// TIA Portal project "Proyecto_Final" (V18)

(* hardware
DEVICE "S7-1500/ET200MP station_1"  S7-1500 station
   slot 0: "Rail_0"  Rack  6ES7 590-1***0-0AA0
   slot 1: "PLC_1"  CPU 1511-1 PN  6ES7 511-1AK00-0AB0  V1.0
      slot 3: "CPU display_1"  6ES7591-1XA00-0AA0
      slot 32768: "PROFINET interface_1"  X1
   slot 2: "CM 1542-5_1"  CM 1542-5  6GK7 542-5DX00-0XE0  V1.0
   slot 3: "DI 16x24VDC HF_1"  DI 16x24VDC HF  6ES7 521-1BH00-0AB0  V1.0
   slot 4: "DQ 16x24VDC/0.5A ST_1"  DQ 16x24VDC/0.5A ST  6ES7 522-1BH00-0AB0  V2.0
   slot 5: "AI 8xU/I/RTD/TC ST_1"  AI 8xU/I/RTD/TC ST  6ES7 531-7KF00-0AB0  V1.0
   slot 6: "AQ 4xU/I ST_1"  AQ 4xU/I ST  6ES7 532-5HD00-0AB0  V1.0
DEVICE "HMI_1"  KTP600 Basic color PN
   slot 0: "HMI_1"  KTP600 Basic color PN  6AV6 647-0AD11-3AX0  12.0.0.0
   slot 1: "HMI_RT_1"  KTP600 Basic color PN  6AV6 647-0AD11-3AX0  12.0.0.0
   slot 5: "HMI_1.IE_CP_1"  PROFINET Interface  12.0.0.0
      slot 1: "PROFINET Interface_1"  PROFINET Interface
         slot 1: "Port_1"  Port
DEVICE "PC-System_1"  SIMATIC PC station
   slot 0: "SIMATIC PC station"  Rail  SIMATIC PC-Station  V1.0
      slot 125: "Stationmanager"  Station_Manager  V6.0.4
   slot 1: "HMI_RT_2"  WinCC RT Advanced  6AV2 104-0xxxx-xxxx  17.0.0.0
      slot 33792: "Computer interface"  Host interface
   slot 2: "IE general_1"  IE General  IE_CP  V8.2.0
      slot 1: "PROFINET interface"  IEGeneral.Interface.8.2.0
*)

// ===== PLC "PLC_1"  CPU 1511-1 PN =====

VAR_GLOBAL   // PLC tag table "Default tag table"
   "Start" AT %M3.4 : Bool;
   "Stop" AT %M3.5 : Bool;
   "PE" AT %M3.6 : Bool;
   "Motor_Banda" AT %Q0.0 : Bool;
   "Variador_Metal" AT %Q0.1 : Bool;
   "V_Presencia" AT %I0.3 : Bool;
   "Reset" AT %M0.0 : Bool;
   "V_Sensor_Metal" AT %I0.4 : Bool;
   "V_Sensor_Vidrio" AT %I0.6 : Bool;
   "V_Galga" AT %IW2 : Int;
   "Medir" AT %M0.1 : Bool;
   "Metal" AT %M0.2 : Bool;
   "Vidrio" AT %M0.3 : Bool;
   "Plastico" AT %M0.4 : Bool;
   "Temp_1s" AT %M0.5 : Bool;
   "T1s_OK" AT %M0.6 : Bool;
   "CTU_Metal" AT %M0.7 : Bool;
   "Metal_OK" AT %M1.0 : Bool;
   "CTU_Vidrio" AT %M1.1 : Bool;
   "Vidrio_OK" AT %M1.2 : Bool;
   "CTU_Plastico" AT %M1.3 : Bool;
   "Plastico_OK" AT %M1.4 : Bool;
   "Temp_Peso" AT %M1.5 : Bool;
   "Temp_Peso_OK" AT %M1.6 : Bool;
   "PID_Pesaje" AT %M1.7 : Bool;
   "Temp_3s" AT %M2.0 : Bool;
   "T3s_OK" AT %M2.1 : Bool;
   "Peso" AT %M2.2 : Bool;
   "Temp_7s" AT %M2.3 : Bool;
   "T7s_OK" AT %M2.4 : Bool;
   "Temp_5s" AT %M2.5 : Bool;
   "T5s_OK" AT %M2.6 : Bool;
   "Temp_Variador" AT %M2.7 : Bool;
   "Temp_Vari_OK" AT %M3.0 : Bool;
   "R_Metal" AT %M3.1 : Bool;
   "R_Vidrio" AT %M3.2 : Bool;
   "R_Plastico" AT %M3.3 : Bool;
   "Piston_Plastico" AT %Q0.2 : Bool;
   "Start_Fisico" AT %I0.0 : Bool;
   "Stop_Fisico" AT %I0.1 : Bool;
   "PE_Fisico" AT %I0.2 : Bool;
   "Start_Pulse" AT %Q0.3 : Bool;
   "En_Pulse" AT %M4.0 : Bool;
   "Low_Pulse_Active" AT %M4.1 : Bool;
   "High_Pulse_Enable" AT %M4.2 : Bool;
   "High_Pulse_Active" AT %M4.3 : Bool;
   "Low_Pulse_Enable" AT %M4.4 : Bool;
   "Count_Metal" AT %QD100 : Real;
   "Count_Vidrio" AT %QD108 : Real;
   "Count_Plastico" AT %QD104 : Real;
   "Alarma_StartNoPresence" AT %Q1.1 : Bool;
   "Alarma_Inicio" AT %Q1.2 : Bool;
   "Alarma_Final" AT %Q1.3 : Bool;
   "Alarma_PE" AT %Q1.0 : Bool;
   "aux" AT %M20.0 : Bool;
   "Start_Fisico_old" AT %M10.4 : Bool;
   "Material_Detectado" AT %Q1.4 : Bool;
   "STP_FIO" AT %I20.1 : Bool;
   "PE_FIO" AT %I20.2 : Bool;
   "START_FIO" AT %I20.0 : Bool;
   "Stop_HMI" AT %M30.1 : Bool;
   "PE_HMI" AT %M30.2 : Bool;
   "START_HMI" AT %M30.3 : Bool;
   "Receta_1" AT %M30.4 : Bool;
   "R1" AT %M30.5 : Bool;
   "R2" AT %M30.6 : Bool;
   "Receta_2" AT %M30.7 : Bool;
END_VAR

DATA_BLOCK "Block_2_DB"   // DB10
{ S7_Optimized_Access := 'TRUE' }
VERSION : 0.1
// stored: InstanceOfName Block_2
"Block_2"
BEGIN
END_DATA_BLOCK

DATA_BLOCK "Block_1_DB"   // DB11
{ S7_Optimized_Access := 'TRUE' }
VERSION : 0.1
// stored: InstanceOfName Grafcet
"Grafcet"
BEGIN
END_DATA_BLOCK

// folder: System blocks/Program resources

DATA_BLOCK "IEC_Timer_0_DB"   // DB1
{ S7_Optimized_Access := 'TRUE' }
AUTHOR : Simatic
FAMILY : IEC
NAME : IEC_TMR
VERSION : 1.0
// stored: InstanceOfName IEC_TIMER
"IEC_TIMER"
BEGIN
END_DATA_BLOCK

DATA_BLOCK "IEC_Counter_0_DB"   // DB2
{ S7_Optimized_Access := 'TRUE' }
AUTHOR : Simatic
FAMILY : IEC
NAME : CNTR
VERSION : 1.0
// stored: InstanceOfName IEC_COUNTER
"IEC_COUNTER"
BEGIN
END_DATA_BLOCK

DATA_BLOCK "IEC_Counter_0_DB_1"   // DB3
{ S7_Optimized_Access := 'TRUE' }
AUTHOR : Simatic
FAMILY : IEC
NAME : CNTR
VERSION : 1.0
// stored: InstanceOfName IEC_COUNTER
"IEC_COUNTER"
BEGIN
END_DATA_BLOCK

DATA_BLOCK "IEC_Counter_0_DB_2"   // DB4
{ S7_Optimized_Access := 'TRUE' }
AUTHOR : Simatic
FAMILY : IEC
NAME : CNTR
VERSION : 1.0
// stored: InstanceOfName IEC_COUNTER
"IEC_COUNTER"
BEGIN
END_DATA_BLOCK

DATA_BLOCK "IEC_Timer_0_DB_1"   // DB5
{ S7_Optimized_Access := 'TRUE' }
AUTHOR : Simatic
FAMILY : IEC
NAME : IEC_TMR
VERSION : 1.0
// stored: InstanceOfName IEC_TIMER
"IEC_TIMER"
BEGIN
END_DATA_BLOCK

DATA_BLOCK "IEC_Timer_0_DB_2"   // DB6
{ S7_Optimized_Access := 'TRUE' }
AUTHOR : Simatic
FAMILY : IEC
NAME : IEC_TMR
VERSION : 1.0
// stored: InstanceOfName IEC_TIMER
"IEC_TIMER"
BEGIN
END_DATA_BLOCK

DATA_BLOCK "IEC_Timer_0_DB_3"   // DB7
{ S7_Optimized_Access := 'TRUE' }
AUTHOR : Simatic
FAMILY : IEC
NAME : IEC_TMR
VERSION : 1.0
// stored: InstanceOfName IEC_TIMER
"IEC_TIMER"
BEGIN
END_DATA_BLOCK

DATA_BLOCK "IEC_Timer_0_DB_4"   // DB8
{ S7_Optimized_Access := 'TRUE' }
AUTHOR : Simatic
FAMILY : IEC
NAME : IEC_TMR
VERSION : 1.0
// stored: InstanceOfName IEC_TIMER
"IEC_TIMER"
BEGIN
END_DATA_BLOCK

DATA_BLOCK "IEC_Timer_0_DB_5"   // DB9
{ S7_Optimized_Access := 'TRUE' }
AUTHOR : Simatic
FAMILY : IEC
NAME : IEC_TMR
VERSION : 1.0
// stored: InstanceOfName IEC_TIMER
"IEC_TIMER"
BEGIN
END_DATA_BLOCK

// folder: (top level)

FUNCTION_BLOCK "Grafcet"   // FB1, GRAPH_PLUS
{ S7_Optimized_Access := 'TRUE' }
VERSION : 0.1
   VAR_INPUT
      OFF_SQ : Bool := false;   // Turn sequence off
      INIT_SQ : Bool := false;   // Set sequence to initial state
      ACK_EF : Bool := false;   // Acknowledge all errors and faults
      S_PREV : Bool := false;   // Output previous step in parameter S_NO
      S_NEXT : Bool := false;   // Indicate next step in parameter S_NO
      SW_AUTO : Bool := false;   // Automatic mode
      SW_TAP : Bool := false;   // Semiautomatic/switch with transition
      SW_TOP : Bool := false;   // Semiautomatic/ignore transition
      SW_MAN : Bool := false;   // Manual mode
      S_SEL : Int := 0;   // Select step to be output to S_NO
      S_ON : Bool := false;   // Activate step indicated in S_NO
      S_OFF : Bool := false;   // Disable step indicated in S_NO
      T_PUSH : Bool := false;   // Enable transition to switch in semi automatic mode
   END_VAR
   VAR_OUTPUT
      S_NO : Int := 0;   // Step number
      S_MORE : Bool := false;   // More steps are available and can be shown in S_NO
      S_ACTIVE : Bool := false;   // Step indicated in S_NO is active
      ERR_FLT : Bool := false;   // Interlock or supervision group error
      AUTO_ON : Bool := false;   // Automatic mode is active
      TAP_ON : Bool := false;   // Semiautomatic mode/step with transition enabled
      TOP_ON : Bool := false;   // Semiautomatic mode/ignore transition enabled
      MAN_ON : Bool := false;   // Manual mode is active
   END_VAR
   VAR
      HMI_INFO : Array[0..8] of UInt;
      IF_PAR : G7_IfParPlus_V2;
      RT_DATA : G7_RTDataPlus_V2;   // Internal data area
      Trans1 : G7_TransitionPlus_V2;   // Transition structure
      Trans5 : G7_TransitionPlus_V2;   // Transition structure
      Trans7 : G7_TransitionPlus_V2;   // Transition structure
      Trans8 : G7_TransitionPlus_V2;   // Transition structure
      Trans9 : G7_TransitionPlus_V2;   // Transition structure
      Trans10 : G7_TransitionPlus_V2;   // Transition structure
      Trans11 : G7_TransitionPlus_V2;   // Transition structure
      Trans12 : G7_TransitionPlus_V2;   // Transition structure
      Trans13 : G7_TransitionPlus_V2;   // Transition structure
      Trans14 : G7_TransitionPlus_V2;   // Transition structure
      Trans15 : G7_TransitionPlus_V2;   // Transition structure
      Trans16 : G7_TransitionPlus_V2;   // Transition structure
      Trans17 : G7_TransitionPlus_V2;   // Transition structure
      Trans18 : G7_TransitionPlus_V2;   // Transition structure
      Trans19 : G7_TransitionPlus_V2;   // Transition structure
      Trans20 : G7_TransitionPlus_V2;   // Transition structure
      Trans21 : G7_TransitionPlus_V2;   // Transition structure
      Trans22 : G7_TransitionPlus_V2;   // Transition structure
      Trans23 : G7_TransitionPlus_V2;   // Transition structure
      Trans24 : G7_TransitionPlus_V2;   // Transition structure
      Trans26 : G7_TransitionPlus_V2;   // Transition structure
      Trans27 : G7_TransitionPlus_V2;   // Transition structure
      Trans28 : G7_TransitionPlus_V2;   // Transition structure
      Trans29 : G7_TransitionPlus_V2;   // Transition structure
      Trans30 : G7_TransitionPlus_V2;   // Transition structure
      Trans31 : G7_TransitionPlus_V2;   // Transition structure
      Reset : G7_StepPlus_V2;   // Step structure
      "Ingreso Botella" : G7_StepPlus_V2;   // Step structure
      Avance_Banda : G7_StepPlus_V2;   // Step structure
      Pesaje : G7_StepPlus_V2;   // Step structure
      Pos_Metal : G7_StepPlus_V2;   // Step structure
      Contenedor_Metal : G7_StepPlus_V2;   // Step structure
      Fin_Ciclo_Metal : G7_StepPlus_V2;   // Step structure
      Pos_Vidrio : G7_StepPlus_V2;   // Step structure
      Contenedor_Vidrio : G7_StepPlus_V2;   // Step structure
      Fin_Ciclo_Vidrio : G7_StepPlus_V2;   // Step structure
      Pos_Plastico : G7_StepPlus_V2;   // Step structure
      Contenedor_Plastico : G7_StepPlus_V2;   // Step structure
      Fin_Ciclo_Plastico : G7_StepPlus_V2;   // Step structure
      Alarmas : G7_StepPlus_V2;   // Step structure
      Step16 : G7_StepPlus_V2;   // Step structure
      Contenedor_Vidrio_1 : G7_StepPlus_V2;   // Step structure
      Alarmas1 : G7_StepPlus_V2;   // Step structure
      Alarmas3 : G7_StepPlus_V2;   // Step structure
      Step20 : G7_StepPlus_V2;   // Step structure
      SINI : Array[0..1] of USInt;
      LSTT : Array[0..25] of USInt;
      ATAJ : Array[0..25] of USInt;
      ATAB : Array[0..25] of USInt;
      PSTT : Array[0..25] of USInt;
      NSTT : Array[0..25] of USInt;
      ASSJ : Array[0..18] of USInt;
      ASSB : Array[0..18] of USInt;
      PTTS : Array[0..18] of USInt;
      NTTS : Array[0..18] of USInt;
      SW_SQTS : Array[0..18] of USInt;
      SWITCH : Array[0..15] of USInt;
      TVX : Array[0..14] of USInt;
      TTX : Array[0..14] of USInt;
      TSX : Array[0..1] of USInt;
      S00X : Array[0..1] of USInt;
      SOFFX : Array[0..1] of USInt;
      SONX : Array[0..1] of USInt;
      SAX : Array[0..1] of USInt;
      SERRX : Array[0..19] of USInt;
      SMX : Array[0..19] of USInt;
      S0X : Array[0..19] of USInt;
      S1X : Array[0..19] of USInt;
      IL_ALARM_INST : Program_Alarm;
      SUP_ALARM_INST : Program_Alarm;
      STEP_TIME_ALARM_INST : Program_Alarm;
      IEC_TIMER_INST : IEC_TIMER;
      TRANSACTION_FLAG : Bool := false;
   END_VAR
   // SINI[0] := 2;
   // LSTT[0] := 255;
   // LSTT[1] := 255;
   // LSTT[2] := 255;
   // LSTT[3] := 255;
   // LSTT[4] := 255;
   // LSTT[5] := 255;
   // LSTT[6] := 255;
   // LSTT[7] := 255;
   // LSTT[8] := 255;
   // LSTT[9] := 1;
   // LSTT[10] := 255;
   // LSTT[11] := 255;
   // LSTT[12] := 1;
   // LSTT[13] := 255;
   // LSTT[14] := 255;
   // LSTT[15] := 255;
   // LSTT[16] := 1;
   // LSTT[17] := 255;
   // LSTT[19] := 255;
   // ATAJ[1] := 1;
   // ATAJ[2] := 2;
   // ATAJ[3] := 3;
   // ATAJ[4] := 4;
   // ATAJ[5] := 5;
   // ATAJ[6] := 6;
   // ATAJ[7] := 7;
   // ATAJ[8] := 8;
   // ATAJ[9] := 9;
   // ATAJ[10] := 10;
   // ATAJ[11] := 11;
   // ATAJ[12] := 12;
   // ATAJ[13] := 13;
   // ATAJ[14] := 14;
   // ATAJ[15] := 15;
   // ATAJ[16] := 16;
   // ATAJ[17] := 17;
   // ATAJ[18] := 18;
   // ATAJ[19] := 19;
   // ATAJ[20] := 20;
   // ATAJ[21] := 21;
   // ATAB[1] := 1;
   // ATAB[2] := 2;
   // ATAB[3] := 4;
   // ATAB[4] := 5;
   // ATAB[5] := 3;
   // ATAB[6] := 22;
   // ATAB[7] := 7;
   // ATAB[8] := 9;
   // ATAB[9] := 8;
   // ATAB[10] := 24;
   // ATAB[11] := 11;
   // ATAB[12] := 13;
   // ATAB[13] := 12;
   // ATAB[14] := 14;
   // ATAB[15] := 15;
   // ATAB[16] := 17;
   // ATAB[17] := 16;
   // ATAB[18] := 18;
   // ATAB[19] := 19;
   // ATAB[20] := 20;
   // ATAB[21] := 21;
   // PSTT[1] := 1;
   // PSTT[2] := 2;
   // PSTT[3] := 3;
   // PSTT[4] := 3;
   // PSTT[5] := 3;
   // PSTT[6] := 4;
   // PSTT[7] := 5;
   // PSTT[8] := 6;
   // PSTT[9] := 6;
   // PSTT[10] := 7;
   // PSTT[11] := 8;
   // PSTT[12] := 9;
   // PSTT[13] := 9;
   // PSTT[14] := 10;
   // PSTT[15] := 11;
   // PSTT[16] := 12;
   // PSTT[17] := 12;
   // PSTT[18] := 13;
   // PSTT[19] := 14;
   // PSTT[20] := 16;
   // PSTT[21] := 17;
   // NSTT[0] := 1;
   // NSTT[1] := 2;
   // NSTT[2] := 3;
   // NSTT[3] := 4;
   // NSTT[4] := 7;
   // NSTT[5] := 10;
   // NSTT[6] := 5;
   // NSTT[7] := 6;
   // NSTT[8] := 13;
   // NSTT[9] := 1;
   // NSTT[10] := 8;
   // NSTT[11] := 9;
   // NSTT[12] := 1;
   // NSTT[13] := 14;
   // NSTT[14] := 11;
   // NSTT[15] := 12;
   // NSTT[16] := 1;
   // NSTT[17] := 17;
   // NSTT[19] := 16;
   // ASSJ[1] := 1;
   // ASSJ[2] := 2;
   // ASSJ[3] := 3;
   // ASSJ[4] := 4;
   // ASSJ[5] := 5;
   // ASSJ[6] := 6;
   // ASSJ[7] := 7;
   // ASSJ[8] := 8;
   // ASSJ[9] := 9;
   // ASSJ[10] := 10;
   // ASSJ[11] := 11;
   // ASSJ[12] := 12;
   // ASSJ[13] := 13;
   // ASSJ[14] := 14;
   // ASSJ[15] := 15;
   // ASSJ[16] := 16;
   // ASSB[1] := 1;
   // ASSB[2] := 2;
   // ASSB[3] := 3;
   // ASSB[4] := 4;
   // ASSB[5] := 5;
   // ASSB[6] := 6;
   // ASSB[7] := 7;
   // ASSB[8] := 8;
   // ASSB[9] := 9;
   // ASSB[10] := 10;
   // ASSB[11] := 11;
   // ASSB[12] := 12;
   // ASSB[13] := 13;
   // ASSB[14] := 14;
   // ASSB[15] := 15;
   // ASSB[16] := 16;
   // PTTS[0] := 255;
   // PTTS[2] := 1;
   // PTTS[3] := 2;
   // PTTS[4] := 3;
   // PTTS[5] := 6;
   // PTTS[6] := 7;
   // PTTS[7] := 4;
   // PTTS[8] := 10;
   // PTTS[9] := 11;
   // PTTS[10] := 5;
   // PTTS[11] := 14;
   // PTTS[12] := 15;
   // PTTS[13] := 8;
   // PTTS[14] := 13;
   // PTTS[15] := 24;
   // PTTS[16] := 19;
   // NTTS[1] := 1;
   // NTTS[2] := 2;
   // NTTS[3] := 3;
   // NTTS[4] := 6;
   // NTTS[5] := 7;
   // NTTS[6] := 9;
   // NTTS[7] := 10;
   // NTTS[8] := 11;
   // NTTS[9] := 12;
   // NTTS[10] := 14;
   // NTTS[11] := 15;
   // NTTS[12] := 16;
   // NTTS[13] := 18;
   // NTTS[14] := 19;
   // NTTS[15] := 25;
   // NTTS[16] := 20;
   // SW_SQTS[4] := 1;
   // SW_SQTS[5] := 2;
   // SW_SQTS[6] := 2;
   // SW_SQTS[7] := 3;
   // SW_SQTS[8] := 4;
   // SW_SQTS[9] := 4;
   // SW_SQTS[10] := 5;
   // SW_SQTS[11] := 5;
   // SW_SQTS[12] := 5;
   // SW_SQTS[13] := 6;
   // SW_SQTS[14] := 7;
   // SW_SQTS[15] := 8;
   // SW_SQTS[16] := 7;
   // TVX[0] := 16#1;
   // TTX[0] := 16#1;
   // TSX[0] := 16#1;
   // S00X[0] := 16#1;
   // SOFFX[0] := 16#1;
   // SONX[0] := 16#1;
   // SAX[0] := 16#1;
   // SERRX[0] := 16#1;
   // SMX[0] := 16#1;
   // S0X[0] := 16#1;
   // S1X[0] := 16#1;
   // LSTT[22] := 255;
   // LSTT[23] := 6;
   // LSTT[24] := 255;
   // LSTT[25] := 9;
   // ATAJ[22] := 22;
   // ATAJ[23] := 23;
   // ATAJ[24] := 24;
   // ATAJ[25] := 25;
   // ATAB[22] := 6;
   // ATAB[23] := 23;
   // ATAB[24] := 10;
   // ATAB[25] := 25;
   // PSTT[22] := 4;
   // PSTT[23] := 18;
   // PSTT[24] := 7;
   // PSTT[25] := 15;
   // NSTT[22] := 18;
   // NSTT[23] := 6;
   // NSTT[24] := 15;
   // NSTT[25] := 9;
   // ASSJ[17] := 17;
   // ASSJ[18] := 18;
   // ASSB[17] := 17;
   // ASSB[18] := 18;
   // PTTS[17] := 17;
   // PTTS[18] := 22;
   // NTTS[17] := 21;
   // NTTS[18] := 23;
   // SW_SQTS[17] := 9;
   // SW_SQTS[18] := 10;
BEGIN
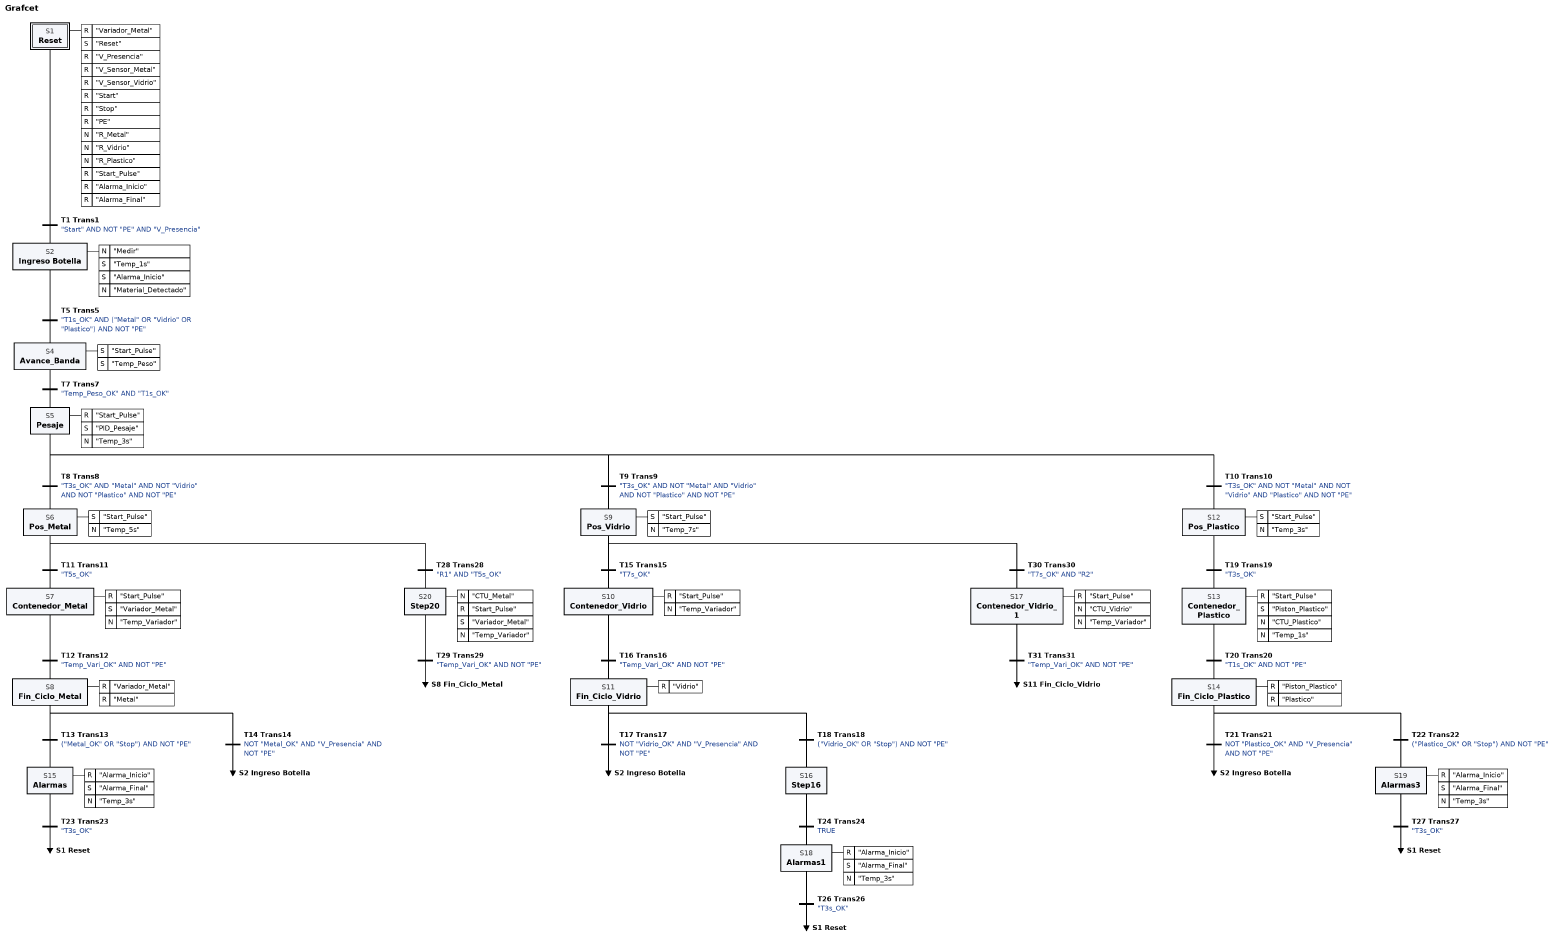
   // sequencer 1
   INITIAL_STEP Reset:   // S1, max time T#10S, warning time T#7S
              R    "Variador_Metal"
              S    "Reset"
              R    "V_Presencia"
              R    "V_Sensor_Metal"
              R    "V_Sensor_Vidrio"
              R    "Start"
              R    "Stop"
              R    "PE"
              N    "R_Metal"
              N    "R_Vidrio"
              N    "R_Plastico"
              R    "Start_Pulse"
              R    "Alarma_Inicio"
              R    "Alarma_Final"
              R    "Receta_1"
              R    "Receta_2"
              R    "R1"
              R    "R2"
   END_STEP
   TRANSITION Trans1 FROM Reset TO "Ingreso Botella"   // T1
      := "Start" AND NOT "PE" AND "V_Presencia";
   END_TRANSITION
   STEP "Ingreso Botella":   // S2, max time T#10S, warning time T#7S
              N    "Medir"
              S    "Temp_1s"
              S    "Alarma_Inicio"
              N    "Material_Detectado"
   END_STEP
   TRANSITION Trans5 FROM "Ingreso Botella" TO Avance_Banda   // T5
      := "T1s_OK" AND ("Metal" OR "Vidrio" OR "Plastico") AND NOT "PE";
   END_TRANSITION
   STEP Avance_Banda:   // S4, max time T#10S, warning time T#7S
              S    "Start_Pulse"
              S    "Temp_Peso"
   END_STEP
   TRANSITION Trans7 FROM Avance_Banda TO Pesaje   // T7
      := "Temp_Peso_OK" AND "T1s_OK";
   END_TRANSITION
   STEP Pesaje:   // S5, max time T#10S, warning time T#7S
              R    "Start_Pulse"
              S    "PID_Pesaje"
              N    "Temp_3s"
   END_STEP
   TRANSITION Trans8 FROM Pesaje TO Pos_Metal   // T8
      := "T3s_OK" AND "Metal" AND NOT "Vidrio" AND NOT "Plastico" AND NOT "PE";
   END_TRANSITION
   TRANSITION Trans9 FROM Pesaje TO Pos_Vidrio   // T9
      := "T3s_OK" AND NOT "Metal" AND "Vidrio" AND NOT "Plastico" AND NOT "PE";
   END_TRANSITION
   TRANSITION Trans10 FROM Pesaje TO Pos_Plastico   // T10
      := "T3s_OK" AND NOT "Metal" AND NOT "Vidrio" AND "Plastico" AND NOT "PE";
   END_TRANSITION
   STEP Pos_Metal:   // S6, max time T#10S, warning time T#7S
              S    "Start_Pulse"
              N    "Temp_5s"
   END_STEP
   TRANSITION Trans11 FROM Pos_Metal TO Contenedor_Metal   // T11
      := "T5s_OK";
   END_TRANSITION
   TRANSITION Trans28 FROM Pos_Metal TO Step20   // T28
      := "R1" AND "T5s_OK";
   END_TRANSITION
   STEP Contenedor_Metal:   // S7, max time T#10S, warning time T#7S
              R    "Start_Pulse"
              S    "Variador_Metal"
              N    "Temp_Variador"
   END_STEP
   TRANSITION Trans12 FROM Contenedor_Metal TO Fin_Ciclo_Metal   // T12
      := "Temp_Vari_OK" AND NOT "PE";
   END_TRANSITION
   STEP Fin_Ciclo_Metal:   // S8, max time T#10S, warning time T#7S
              R    "Variador_Metal"
              R    "Metal"
   END_STEP
   TRANSITION Trans13 FROM Fin_Ciclo_Metal TO Alarmas   // T13
      := ("Metal_OK" OR "Stop") AND NOT "PE";
   END_TRANSITION
   TRANSITION Trans14 FROM Fin_Ciclo_Metal TO "Ingreso Botella"   // T14, jump
      := NOT "Metal_OK" AND "V_Presencia" AND NOT "PE";
   END_TRANSITION
   STEP Pos_Vidrio:   // S9, max time T#10S, warning time T#7S
              S    "Start_Pulse"
              N    "Temp_7s"
   END_STEP
   TRANSITION Trans15 FROM Pos_Vidrio TO Contenedor_Vidrio   // T15
      := "T7s_OK";
   END_TRANSITION
   TRANSITION Trans30 FROM Pos_Vidrio TO Contenedor_Vidrio_1   // T30
      := "T7s_OK" AND "R2";
   END_TRANSITION
   STEP Contenedor_Vidrio:   // S10, max time T#10S, warning time T#7S
              R    "Start_Pulse"
              N    "Temp_Variador"
   END_STEP
   TRANSITION Trans16 FROM Contenedor_Vidrio TO Fin_Ciclo_Vidrio   // T16
      := "Temp_Vari_OK" AND NOT "PE";
   END_TRANSITION
   STEP Fin_Ciclo_Vidrio:   // S11, max time T#10S, warning time T#7S
              R    "Vidrio"
   END_STEP
   TRANSITION Trans17 FROM Fin_Ciclo_Vidrio TO "Ingreso Botella"   // T17, jump
      := NOT "Vidrio_OK" AND "V_Presencia" AND NOT "PE";
   END_TRANSITION
   TRANSITION Trans18 FROM Fin_Ciclo_Vidrio TO Step16   // T18
      := ("Vidrio_OK" OR "Stop") AND NOT "PE";
   END_TRANSITION
   STEP Pos_Plastico:   // S12, max time T#10S, warning time T#7S
              S    "Start_Pulse"
              N    "Temp_3s"
   END_STEP
   TRANSITION Trans19 FROM Pos_Plastico TO Contenedor_Plastico   // T19
      := "T3s_OK";
   END_TRANSITION
   STEP Contenedor_Plastico:   // S13, max time T#10S, warning time T#7S
              R    "Start_Pulse"
              S    "Piston_Plastico"
              N    "CTU_Plastico"
              N    "Temp_1s"
   END_STEP
   TRANSITION Trans20 FROM Contenedor_Plastico TO Fin_Ciclo_Plastico   // T20
      := "T1s_OK" AND NOT "PE";
   END_TRANSITION
   STEP Fin_Ciclo_Plastico:   // S14, max time T#10S, warning time T#7S
              R    "Piston_Plastico"
              R    "Plastico"
   END_STEP
   TRANSITION Trans21 FROM Fin_Ciclo_Plastico TO "Ingreso Botella"   // T21, jump
      := NOT "Plastico_OK" AND "V_Presencia" AND NOT "PE";
   END_TRANSITION
   TRANSITION Trans22 FROM Fin_Ciclo_Plastico TO Alarmas3   // T22
      := ("Plastico_OK" OR "Stop") AND NOT "PE";
   END_TRANSITION
   STEP Alarmas:   // S15, max time T#10S, warning time T#7S
              R    "Alarma_Inicio"
              S    "Alarma_Final"
              N    "Temp_3s"
   END_STEP
   TRANSITION Trans23 FROM Alarmas TO Reset   // T23, jump
      := "T3s_OK";
   END_TRANSITION
   STEP Step16:   // S16, max time T#10S, warning time T#7S
   END_STEP
   TRANSITION Trans24 FROM Step16 TO Alarmas1   // T24
      := TRUE;
   END_TRANSITION
   STEP Alarmas1:   // S18, max time T#10S, warning time T#7S
              R    "Alarma_Inicio"
              S    "Alarma_Final"
              N    "Temp_3s"
   END_STEP
   TRANSITION Trans26 FROM Alarmas1 TO Reset   // T26, jump
      := "T3s_OK";
   END_TRANSITION
   STEP Alarmas3:   // S19, max time T#10S, warning time T#7S
              R    "Alarma_Inicio"
              S    "Alarma_Final"
              N    "Temp_3s"
   END_STEP
   TRANSITION Trans27 FROM Alarmas3 TO Reset   // T27, jump
      := "T3s_OK";
   END_TRANSITION
   STEP Step20:   // S20, max time T#10S, warning time T#7S
              N    "CTU_Metal"
              R    "Start_Pulse"
              S    "Variador_Metal"
              N    "Temp_Variador"
   END_STEP
   TRANSITION Trans29 FROM Step20 TO Fin_Ciclo_Metal   // T29, jump
      := "Temp_Vari_OK" AND NOT "PE";
   END_TRANSITION
   STEP Contenedor_Vidrio_1:   // S17, max time T#10S, warning time T#7S
              R    "Start_Pulse"
              N    "CTU_Vidrio"
              N    "Temp_Variador"
   END_STEP
   TRANSITION Trans31 FROM Contenedor_Vidrio_1 TO Fin_Ciclo_Vidrio   // T31, jump
      := "Temp_Vari_OK" AND NOT "PE";
   END_TRANSITION
END_FUNCTION_BLOCK

FUNCTION_BLOCK "Block_2"   // FB2, STL
{ S7_Optimized_Access := 'TRUE' }
VERSION : 0.1
   VAR
      IEC_Timer_0_Instance : TON_LTIME;
      DB1 : TON_LTIME;
   END_VAR
BEGIN

REGION Network 1
   // Habilitación
         A     "Start_Pulse";
         =     "En_Pulse";

   // Enable T1
         A     "En_Pulse";
         AN    "Low_Pulse_Active";
         =     "High_Pulse_Enable";

         CALL  #DB1
         ( IN := "High_Pulse_Enable",
           PT := LT#25000ns,
           Q  := "High_Pulse_Active",
           ET :=
         );


   // Enable T2
         A     "En_Pulse";
         A     "High_Pulse_Active";
         =     "Low_Pulse_Enable";

         CALL  #IEC_Timer_0_Instance
         ( IN := "Low_Pulse_Enable",
           PT := LT#25000ns,
           Q  := "Low_Pulse_Active",
           ET :=
         );

   // Salida
         A     "High_Pulse_Active";
         =     "Motor_Banda";
END_REGION
END_FUNCTION_BLOCK

ORGANIZATION_BLOCK "Main"   // OB1, LAD, ProgramCycle
TITLE = "Main Program Sweep (Cycle)"
{ S7_Optimized_Access := 'TRUE' }
VERSION : 0.1
   VAR_INPUT
      Initial_Call : Bool;   // Initial call of this OB
      Remanence : Bool;   // =True, if remanent data are available
   END_VAR
BEGIN

REGION Network 1
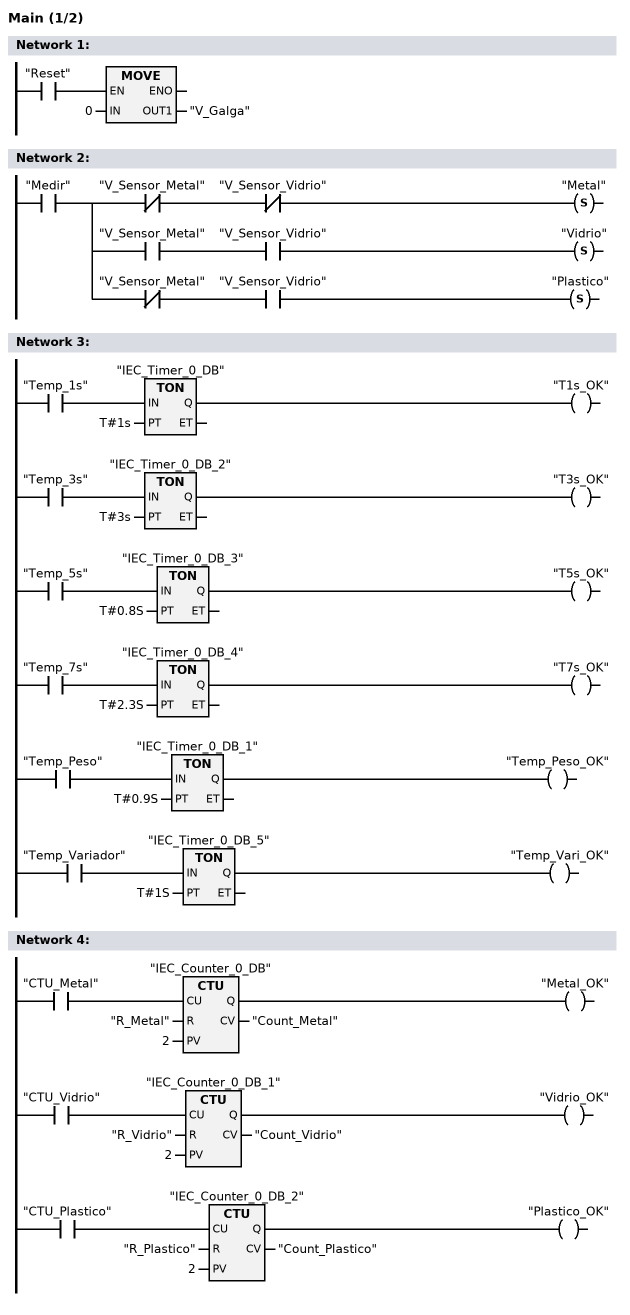
   RUNG wire#powerrail
      Contact( "Reset" )
      Move(in := 0, out1 => "V_Galga")
   END_RUNG
   // the same network as SCL:
   IF "Reset" THEN "V_Galga" := 0; END_IF;
END_REGION

REGION Network 2
   RUNG wire#powerrail
      Contact( "Medir" )
      wire#w1
      I_Contact( "V_Sensor_Metal" )
      I_Contact( "V_Sensor_Vidrio" )
      S_Coil( "Metal" )
   END_RUNG
   RUNG wire#w1
      Contact( "V_Sensor_Metal" )
      Contact( "V_Sensor_Vidrio" )
      S_Coil( "Vidrio" )
   END_RUNG
   RUNG wire#w1
      I_Contact( "V_Sensor_Metal" )
      Contact( "V_Sensor_Vidrio" )
      S_Coil( "Plastico" )
   END_RUNG
   // the same network as SCL:
   IF "Medir" AND NOT "V_Sensor_Metal" AND NOT "V_Sensor_Vidrio" THEN "Metal" := TRUE; END_IF;
   IF "Medir" AND "V_Sensor_Metal" AND "V_Sensor_Vidrio" THEN "Vidrio" := TRUE; END_IF;
   IF "Medir" AND NOT "V_Sensor_Metal" AND "V_Sensor_Vidrio" THEN "Plastico" := TRUE; END_IF;
END_REGION

REGION Network 3
   "IEC_Timer_0_DB".TON(IN := "Temp_1s", PT := T#1s);
   "T1s_OK" := "IEC_Timer_0_DB".Q;
   "IEC_Timer_0_DB_2".TON(IN := "Temp_3s", PT := T#3s);
   "T3s_OK" := "IEC_Timer_0_DB_2".Q;
   "IEC_Timer_0_DB_3".TON(IN := "Temp_5s", PT := T#0.8S);
   "T5s_OK" := "IEC_Timer_0_DB_3".Q;
   "IEC_Timer_0_DB_4".TON(IN := "Temp_7s", PT := T#2.3S);
   "T7s_OK" := "IEC_Timer_0_DB_4".Q;
   "IEC_Timer_0_DB_1".TON(IN := "Temp_Peso", PT := T#0.9S);
   "Temp_Peso_OK" := "IEC_Timer_0_DB_1".Q;
   "IEC_Timer_0_DB_5".TON(IN := "Temp_Variador", PT := T#1S);
   "Temp_Vari_OK" := "IEC_Timer_0_DB_5".Q;
END_REGION

REGION Network 4
   "IEC_Counter_0_DB".CTU(CU := "CTU_Metal", R := "R_Metal", PV := 2, CV => "Count_Metal");
   "Metal_OK" := "IEC_Counter_0_DB".Q;
   "IEC_Counter_0_DB_1".CTU(CU := "CTU_Vidrio", R := "R_Vidrio", PV := 2, CV => "Count_Vidrio");
   "Vidrio_OK" := "IEC_Counter_0_DB_1".Q;
   "IEC_Counter_0_DB_2".CTU(CU := "CTU_Plastico", R := "R_Plastico", PV := 2, CV => "Count_Plastico");
   "Plastico_OK" := "IEC_Counter_0_DB_2".Q;
END_REGION

REGION Network 5
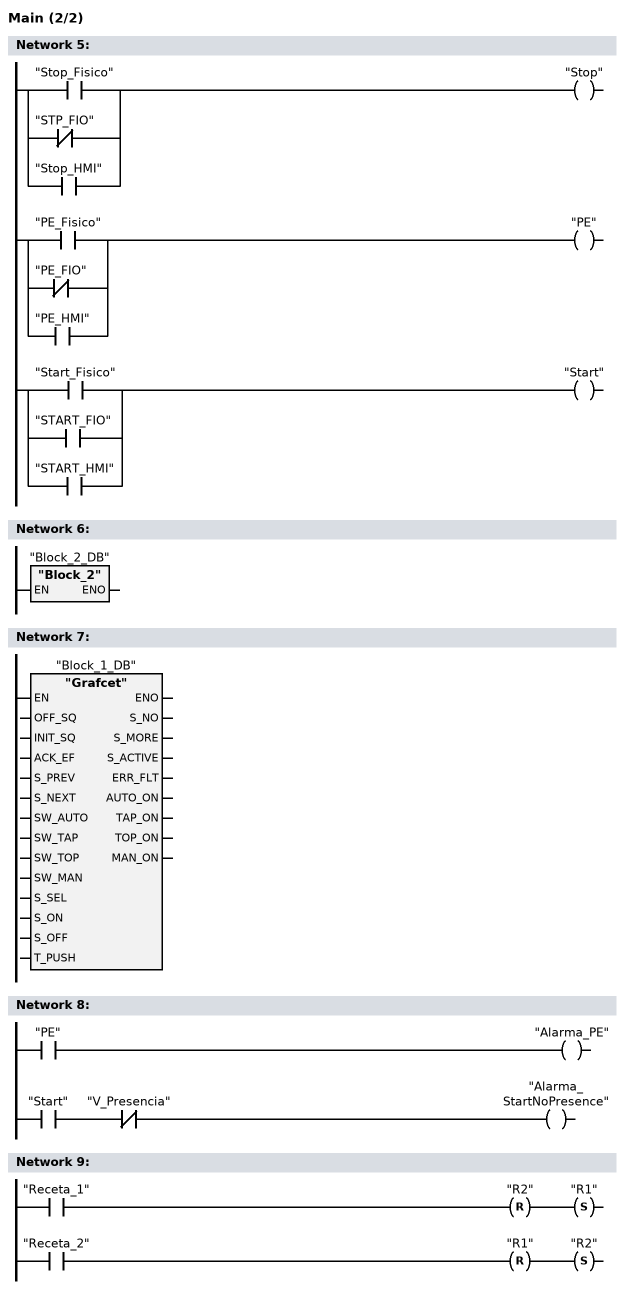
   RUNG wire#powerrail
      Contact( "Stop_Fisico" )
      wire#w1
      Coil( "Stop" )
   END_RUNG
   RUNG wire#powerrail
      I_Contact( "STP_FIO" )
   END_RUNG wire#w1
   RUNG wire#powerrail
      Contact( "Stop_HMI" )
   END_RUNG wire#w1
   RUNG wire#powerrail
      Contact( "PE_Fisico" )
      wire#w2
      Coil( "PE" )
   END_RUNG
   RUNG wire#powerrail
      I_Contact( "PE_FIO" )
   END_RUNG wire#w2
   RUNG wire#powerrail
      Contact( "PE_HMI" )
   END_RUNG wire#w2
   RUNG wire#powerrail
      Contact( "Start_Fisico" )
      wire#w3
      Coil( "Start" )
   END_RUNG
   RUNG wire#powerrail
      Contact( "START_FIO" )
   END_RUNG wire#w3
   RUNG wire#powerrail
      Contact( "START_HMI" )
   END_RUNG wire#w3
   // the same network as SCL:
   "Stop" := "Stop_Fisico" OR NOT "STP_FIO" OR "Stop_HMI";
   "PE" := "PE_Fisico" OR NOT "PE_FIO" OR "PE_HMI";
   "Start" := "Start_Fisico" OR "START_FIO" OR "START_HMI";
END_REGION

REGION Network 6
   RUNG wire#powerrail
      "Block_2_DB"()
   END_RUNG
   // the same network as SCL:
   "Block_2_DB"();   // "Block_2"
END_REGION

REGION Network 7
   RUNG wire#powerrail
      "Block_1_DB"(OFF_SQ :=, INIT_SQ :=, ACK_EF :=, S_PREV :=, S_NEXT :=, SW_AUTO :=, SW_TAP :=, SW_TOP :=, SW_MAN :=, S_SEL :=, S_ON :=, S_OFF :=, T_PUSH :=, S_NO =>, S_MORE =>, S_ACTIVE =>, ERR_FLT =>, AUTO_ON =>, TAP_ON =>, TOP_ON =>, MAN_ON =>)
   END_RUNG
   // the same network as SCL:
   "Block_1_DB"();   // "Grafcet"
END_REGION

REGION Network 8
   RUNG wire#powerrail
      Contact( "PE" )
      Coil( "Alarma_PE" )
   END_RUNG
   RUNG wire#powerrail
      Contact( "Start" )
      I_Contact( "V_Presencia" )
      Coil( "Alarma_StartNoPresence" )
   END_RUNG
   // the same network as SCL:
   "Alarma_PE" := "PE";
   "Alarma_StartNoPresence" := "Start" AND NOT "V_Presencia";
END_REGION

REGION Network 9
   RUNG wire#powerrail
      Contact( "Receta_1" )
      R_Coil( "R2" )
      S_Coil( "R1" )
   END_RUNG
   RUNG wire#powerrail
      Contact( "Receta_2" )
      R_Coil( "R1" )
      S_Coil( "R2" )
   END_RUNG
   // the same network as SCL:
   IF "Receta_1" THEN
       "R2" := FALSE;
       "R1" := TRUE;
   END_IF;
   IF "Receta_2" THEN
       "R1" := FALSE;
       "R2" := TRUE;
   END_IF;
END_REGION
END_ORGANIZATION_BLOCK

(* ===== HMI "HMI_RT_1" =====
system functions are stored by id; their names below are inferred from use
connection "HMI_Connection_1": ETHERNET, SMART_S7_1500_OMS

HMI tags "Default tag table"
   "Count_Metal" : Real = PLC Count_Metal AT %QD100, 1 s
   "Count_Vidrio" : Real = PLC Count_Vidrio AT %QD108, 1 s
   "Alarma_StartNoPresence" : Bool = PLC Alarma_StartNoPresence AT %Q1.1, 1 s
   "Alarma_Final" : Bool = PLC Alarma_Final AT %Q1.3, 1 s
   "Alarma_Inicio" : Bool = PLC Alarma_Inicio AT %Q1.2, 1 s
   "Alarma_PE" : Bool = PLC Alarma_PE AT %Q1.0, 1 s
   "Start_Pulse" : Bool = PLC Start_Pulse AT %Q0.3, 1 s
   "START_HMI" : Bool = PLC START_HMI AT %M30.3, 1 s
   "Stop_HMI" : Bool = PLC Stop_HMI AT %M30.1, 1 s
   "PE_HMI" : Bool = PLC PE_HMI AT %M30.2, 1 s
   "Receta_1" : Bool = PLC Receta_1 AT %M30.4, 1 s
   "Receta_2" : Bool = PLC Receta_2 AT %M30.7, 1 s
   "R2" : Bool = PLC R2 AT %M30.6, 1 s
   "R1" : Bool = PLC R1 AT %M30.5, 1 s

screen "Root screen" 320x240, template "Template_1"
   GraphicView "Graphic view_1" at 0,0 size 320x240; Picture "WhatsApp Image 2026-05-28 at 09.53.20"
   Button "Screen0" at 214,207 size 104x30; TextOff 'Proceso'; TextOn 'Screen0'
      on Release: ActivateScreen("Screen0", 0)

screen "Screen0" 320x240, template "Template_1"
   Button "Back" at 1,1 size 104x30; TextOff 'Back'
      on Release: ActivateScreen("Root screen", 0)
   Button "Screen1" at 106,1 size 104x30; TextOff 'Recetas'; TextOn 'Screen1'
      on Release: ActivateScreen("Screen1", 0)
   GraphicView "Graphic view_2" at 16,49 size 71x55; Picture "Graphic_2"
      Visibility <- "Start_Pulse"
   GraphicView "Graphic view_1" at 16,49 size 73x51; Picture "Graphic_1"
      Visibility <- "Start_Pulse"
   Button "Button_1" at 10,202 size 96x32; TextOff 'START'
      Appearance <- "START_HMI"
   Button "Button_2" at 116,202 size 96x32; TextOn 'STOP'; TextOff 'STOP'
      Appearance <- "Stop_HMI"
   Button "Button_3" at 223,202 size 96x32; TextOn 'PE'; TextOff 'PE'
      Appearance <- "PE_HMI"
   GraphicView "Graphic view_3" at 242,26 size 78x79; Picture "imagen_2026-05-29_080438939"
   GraphicView "Graphic view_4" at 200,37 size 70x67; Picture "imagen_2026-05-29_080314886"
   GraphicView "Graphic view_6" at 0,160 size 319x42; Picture "Graphic_4"
   GraphicView "Graphic view_5" at 36,126 size 27x55; Picture "Graphic_5"
   IOField "I/O field_1" at 200,105 size 56x23; FormatPattern 999
      Appearance <- "Count_Metal"
   IOField "I/O field_2" at 264,105 size 56x23; FormatPattern 999
      Appearance <- "Count_Vidrio"
   Circle "Circle_3" at 116,74 size 24x24
      Appearance <- "R2"
   TextField "Text field_1" at 124,45 size 16x13; Text 'R1'
      Appearance <- "R1"
   TextField "Text field_2" at 124,78 size 16x13; Text 'R2'
   IOField "I/O field_3" at 256,8 size 56x23; FormatPattern 999
      Appearance <- "Count_Vidrio"
   TextField "Text field_5" at 222,10 size 32x13; Text 'PESO:'

screen "Screen1" 320x240, template "Template_1"
   Button "Back" at 1,1 size 104x30; TextOff 'Back'
      on Release: ActivateScreen("Screen0", 0)
   Button "Back_1" at 113,1 size 104x30; TextOn 'Back'; TextOff 'Home'
      on Release: ActivateScreen("Root screen", 0)
   Button "Button_1" at 211,40 size 96x32; TextOff 'Receta 1'
      on Press: InvertBit("Receta_1")
   Button "Button_2" at 211,72 size 96x32; TextOff 'Receta 2'
      on Press: InvertBit("Receta_2")
   Circle "Circle_1" at 12,36 size 48x48
      Appearance <- "Alarma_StartNoPresence"
   Circle "Circle_2" at 12,90 size 48x48
      Appearance <- "Alarma_Final"
   Circle "Circle_3" at 12,139 size 48x48
      Appearance <- "Alarma_Inicio"
   Circle "Circle_4" at 12,188 size 48x48
      Appearance <- "Alarma_PE"
   TextField "Text field_1" at 73,48 size 91x16; Text 'SIN MATERIAL'
   TextField "Text field_2" at 72,103 size 37x16; Text 'FINAL'
   TextField "Text field_3" at 68,156 size 81x16; Text 'Alarma Inicio'
   TextField "Text field_4" at 72,200 size 140x16; Text 'PARO DE EMERGENCIA'
*)

(* ===== HMI "HMI_RT_2" =====
system functions are stored by id; their names below are inferred from use
connection "HMI_Connection_2": ETHERNET, S7_1500_OMS

HMI tags "Default tag table"
   "Start" : Bool = PLC Start AT %M3.4, 1 s
   "PE" : Bool = PLC PE AT %M3.6, 1 s
   "Stop" : Bool = PLC Stop AT %M3.5, 1 s
   "Start_Pulse" : Bool = PLC Start_Pulse AT %Q0.3, 1 s
   "Metal" : Bool = PLC Metal AT %M0.2, 1 s
   "Vidrio" : Bool = PLC Vidrio AT %M0.3, 1 s
   "Plastico" : Bool = PLC Plastico AT %M0.4, 1 s
   "Count_Metal" : Real = PLC Count_Metal AT %QD100, 1 s
   "Count_Vidrio" : Real = PLC Count_Vidrio AT %QD108, 1 s
   "Count_Plastico" : Real = PLC Count_Plastico AT %QD104, 1 s
   "Metal_OK" : Bool = PLC Metal_OK AT %M1.0, 1 s
   "Vidrio_OK" : Bool = PLC Vidrio_OK AT %M1.2, 1 s
   "Plastico_OK" : Bool = PLC Plastico_OK AT %M1.4, 1 s
   "Alarma_Inicio" : Bool = PLC Alarma_Inicio AT %Q1.2, 1 s
   "Alarma_PE" : Bool = PLC Alarma_PE AT %Q1.0, 1 s
   "Alarma_StartNoPresence" : Bool = PLC Alarma_StartNoPresence AT %Q1.1, 1 s
   "Alarma_Final" : Bool = PLC Alarma_Final AT %Q1.3, 1 s

screen "Screen_1" 1024x768
   GraphicView "Graphic view_7" at 535,470 size 187x105; Picture "Graphic_8"
      Visibility <- "Start_Pulse"
   GraphicView "Graphic view_1" at 9,39 size 393x242; Picture "WhatsApp Image 2026-05-28 at 09.53.20"
   TextField "Text field_1" at 83,7 size 249x29; Text 'Calsificador de Botellas'
   Rectangle "Rectangle_1" at 409,39 size 67x37
      Appearance <- "Start"
   TextField "Text field_2" at 422,46 size 43x22; Text 'Start'
   Rectangle "Rectangle_2" at 409,89 size 67x37
      Appearance <- "Stop"
   TextField "Text field_3" at 422,96 size 39x22; Text 'Stop'
   Rectangle "Rectangle_3" at 409,137 size 119x55
      Appearance <- "PE"
   TextField "Text field_4" at 422,144 size 92x40; Text 'Paro de Emergencia'
   Circle "Circle_1" at 67,302 size 52x52
      Appearance <- "Start_Pulse"
   TextField "Text field_5" at 46,361 size 99x22; Text 'Motor Banda'
   GraphicView "Graphic view_2" at 152,306 size 96x102; Picture "imagen_2026-05-29_080314886"
   GraphicView "Graphic view_3" at 355,302 size 96x104; Picture "plastico"
   GraphicView "Graphic view_4" at 256,302 size 96x109; Picture "imagen_2026-05-29_080438939"
   TextField "Text field_6" at 176,411 size 47x22; Text 'Metal'
   TextField "Text field_7" at 279,412 size 50x22; Text 'Vidrio'
   TextField "Text field_8" at 374,412 size 65x22; Text 'Plastico'
   Circle "Circle_2" at 184,436 size 32x32
      Appearance <- "Metal"
   Circle "Circle_3" at 292,436 size 32x32
      Appearance <- "Vidrio"
   Circle "Circle_4" at 392,435 size 32x32
      Appearance <- "Plastico"
   IOField "I/O field_1" at 152,483 size 96x32; FormatPattern s99999
      ProcessValue <- "Count_Metal"
   IOField "I/O field_2" at 259,483 size 96x32; FormatPattern s99999
      ProcessValue <- "Count_Vidrio"
   IOField "I/O field_3" at 366,483 size 96x32; FormatPattern s99999
      ProcessValue <- "Count_Plastico"
   TextField "Text field_9" at 45,488 size 95x22; Text 'Contadores:'
   TextField "Text field_10" at 44,535 size 96x40; Text 'Receta completada:'
   Circle "Circle_5" at 184,537 size 32x32
      Appearance <- "Metal_OK"
   Circle "Circle_6" at 294,534 size 32x32
      Appearance <- "Vidrio_OK"
   Circle "Circle_7" at 404,531 size 32x32
      Appearance <- "Plastico_OK"
   Circle "Circle_8" at 575,247 size 48x48
      Appearance <- "Alarma_Inicio"
   TextField "Text field_11" at 549,211 size 71x22; Text 'Alarmas:'
   TextField "Text field_12" at 574,297 size 48x22; Text 'Inicio'
   Circle "Circle_9" at 675,247 size 48x48
      Appearance <- "Alarma_PE"
   TextField "Text field_13" at 687,297 size 24x22; Text 'PE'
   Circle "Circle_10" at 677,327 size 48x48
      Appearance <- "Alarma_Final"
   TextField "Text field_14" at 680,377 size 42x22; Text 'Final'
   Circle "Circle_11" at 577,325 size 48x48
      Appearance <- "Alarma_StartNoPresence"
   TextField "Text field_15" at 551,377 size 96x22; Text 'Sin Material'
   GraphicView "Graphic view_5" at 0,654 size 923x99; Picture "Graphic_4"
   GraphicView "Graphic view_6" at 152,602 size 35x95; Picture "Graphic_5"
   GraphicView "Graphic view_8" at 535,470 size 187x105; Picture "Graphic_7"
      Visibility <- "Start_Pulse"
   Button "Button_1" at 508,43 size 96x32; TextOff 'START'
      on Press: InvertBit("Start")
   Button "Button_2" at 508,86 size 96x32; TextOff 'STOP'
      on Press: InvertBit("Stop")
   Button "Button_3" at 538,150 size 96x32; TextOff 'PE'
      on Press: InvertBit("PE")
*)